VISUALIZATION VISU_Robot  // 800x480
END_VISUALIZATION

(* stored: Version 1.1.0.1, ProductVersion 3.1.4026.18
   Visu VISU_Robot: Id {375c1ba1-7b6d-4f7b-85ad-63ff328f17e3} *)
